SUBAPPLICATION mapping_Uebung_031 (* LED Strip *)
  (* Standard: 61499-2 *)
  (* Version 1.0, 2023-10-23, franz *)
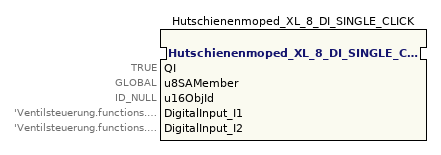
  FBS
    Hutschienenmoped_XL_8_DI_SINGLE_CLICK : Hutschienenmoped_XL_8_DI_SINGLE_CLICK(QI := TRUE, u8SAMember := GLOBAL, u16ObjId := ID_NULL, DigitalInput_I1 := 'Ventilsteuerung.functions.DigitalInput_I1_CLK', DigitalInput_I2 := 'Ventilsteuerung.functions.DigitalInput_I2_CLK');
  END_FBS
END_SUBAPPLICATION
